# EPICS substitutions: apps/svtCtrlApp/Db/svtOnOff.substitutions
file "db/svtOnOff-1side.db" {
pattern { SIDE ONOFF }
{ T OFF }
{ B OFF }
}

file "db/svtOnOff-1reg.db" {
pattern { REG ONOFF }
{ 1 OFF }
{ 2 OFF }
{ 3 OFF }
}

file "db/svtOnOff-1type.db" {
pattern { TYPE ONOFF }
{ HV OFF }
}
